INTERFACE I_ModeManager

METHOD AddCustomPackMode : BOOL
VAR_INPUT
  index : UINT;
  newPackMode : I_PackMode;
END_VAR
END_METHOD

METHOD AddPackModes : BOOL
VAR_INPUT
  prodMode : I_PackMode;
  maintMode : I_PackMode;
  manMode : I_PackMode;
END_VAR
END_METHOD

METHOD PUBLIC AddStateModule
VAR_INPUT
  stateModule : I_StateModule;
END_VAR
END_METHOD

METHOD PUBLIC ChangeMode
VAR_INPUT
  Mode : E_PMLUnitMode;
END_VAR
END_METHOD

PROPERTY PUBLIC CommandedMode : E_PMLProtectedUnitMode
GET
END_GET
END_PROPERTY

PROPERTY CurrentMode : E_PMLProtectedUnitMode
GET
END_GET
END_PROPERTY

METHOD PUBLIC CyclicLogic
VAR_INPUT
END_VAR
END_METHOD

PROPERTY PUBLIC LogModeChanges : BOOL
GET
END_GET
SET
END_SET
END_PROPERTY

PROPERTY PUBLIC  ModeNames : REFERENCE TO ARRAY[0..31] OF STRING
GET
END_GET
END_PROPERTY

END_INTERFACE

(* stored: Version 1.1.0.1, ProductVersion 3.1.4024.12
   Itf I_ModeManager: Id {43f4dfa9-aee4-40ad-83ad-b4f8b760fd6a}
   Folder Properties: Id {bf5fc7df-2960-4dc8-b341-f3e0c472a979}
   Folder Public: Id {ecae9b5b-a7d7-4888-b825-b1ed99b3e70f}
   Method AddCustomPackMode: Id {9bdf90f7-a39c-4a84-904e-d7ee32768723}
   Method AddPackModes: Id {b5ed3537-a540-4df6-aa09-1c86491aefd3}
   Method AddStateModule: Id {73dd2db3-ea8a-4c53-a2cb-51cd0facaf63}
   Method ChangeMode: Id {341d4751-712a-4607-9d66-147759d82e06}
   Property CommandedMode: Id {533c7242-61a5-4641-9c71-744c83e164ae}
   Get Get: Id {c94a2607-4f3d-4750-9311-512034603189}
   Property CurrentMode: Id {a9806cdd-9a75-41f3-8d95-823cb649c948}
   Get Get: Id {07bfa944-506d-4241-973c-68128961a3d2}
   Method CyclicLogic: Id {d6747437-05f6-4ad7-9c36-359e1d42e79b}
   Property LogModeChanges: Id {a4016744-9cd6-40e1-87b9-41eff92c47c6}
   Get Get: Id {b1d41291-8a9e-4993-982a-980db0d5409f}
   Set Set: Id {1e3d322e-6260-4d5a-853d-6dc59abbdc95}
   Property ModeNames: Id {46040903-c3d9-465c-9405-a19d3141468c}
   Get Get: Id {b2b22703-b975-4696-8b83-2e5313ce89c4} *)
